// TIA Portal V17 export
// export: Created 2022-04-06T07:28:39.8526762Z, ExportSetting WithDefaults, DisplayName Totally Integrated Automation Portal, DisplayVersion V17, DisplayName TIA Portal Openness, DisplayVersion V17, DisplayName TIA Portal Version Control Interface, DisplayVersion V17, DisplayName TIA Portal Test Suite Advanced, DisplayVersion V17, DisplayName SINAMICS Startdrive Advanced, DisplayVersion V17, DisplayName SINAMICS Startdrive G130, G150, S120, S150, SINAMICS MV, S210, DisplayVersion V17, DisplayName SINAMICS Startdrive G110M, G120, G120C, G120D, G120P, G115D, DisplayVersion V17, DisplayName STEP 7 Professional, DisplayVersion V17, DisplayName STEP 7 Safety, DisplayVersion V17, DisplayName WinCC Advanced / Unified PC, DisplayVersion V17
DATA_BLOCK "TestSclDb"   // DB7
{ S7_Optimized_Access := 'TRUE' }
VERSION : 0.1
// stored: AutoNumber true, DBAccessibleFromOPCUA true, DBAccessibleFromWebserver true, IsOnlyStoredInLoadMemory false, IsRetainMemResEnabled false, IsWriteProtectedInAS false, MemoryReserve 100
   VAR
      start : Bool;
      state1 : Bool;
      state2 : Bool;
      state3 : Bool;
      state4 : Bool;
      state5 : Bool;
      state6 : Bool;
      nextStep : Bool;
      cond1 : Int;
      testCond1 : Bool;
      result : Bool;
      aArray : Array[0..9] of Int;
      bArray : Array[0..9] of Int;
      count : SInt := 9;
      string1 : Array[0..10] of String[50];
      string2 : Array[0..10] of String[50];
      string3 : Array[0..10] of String[50];
      dumpString : String;
   END_VAR
BEGIN
   bArray[0] := 1;
END_DATA_BLOCK
